TYPE T_Ctrl_SIf_CYL_Ilk :
STRUCT
	///interlock retraction of cylinder
	bolRetract: BOOL;
	///interlock extend of cylinder
	bolExtend: BOOL;
END_STRUCT
END_TYPE

(* stored: Version 1.1.0.1, ProductVersion 3.1.0.19
   DUT T_Ctrl_SIf_CYL_Ilk: Id {306d491c-702b-4109-95c1-9e9e92b5c7b7} *)
